{attribute addProperty BoxType "EL3632-0000-0016"}
{attribute addProperty Id "STATUSAT %I*STATUS_F9B4A013162"}
{attribute addProperty CRC "364138195"}
{attribute addProperty SizeInBites "16"}
{attribute addProperty SizeInBytes "2"}
TYPE Ch2_Status_15B44ED3 :
STRUCT
	{attribute addProperty Name "STATUS"}
	STATUS AT %I* : STATUS_F9B4A013;
END_STRUCT
END_TYPE

(* stored: Version 1.2.0.0, ProductVersion 3.1.4024.9
   DUT Ch2_Status_15B44ED3: Id {8792589b-a7b8-4f40-aa0b-bb6e334a2aec} *)
